PROGRAM LateBlanking_Temperature
VAR
	P3_FB_Temperature: ARRAY[1..104] OF FB_Temperature;
	i:INT;
END_VAR

ACT2();

IF Tem_HOT THEN
arrTempCtrl[1].Out.PIDRun:=TRUE;
arrTempCtrl[2].Out.PIDRun:=TRUE;
arrTempCtrl[3].Out.PIDRun:=TRUE;
arrTempCtrl[4].Out.PIDRun:=TRUE;
arrTempCtrl[5].Out.PIDRun:=TRUE;
arrTempCtrl[6].Out.PIDRun:=TRUE;
arrTempCtrl[7].Out.PIDRun:=TRUE;
arrTempCtrl[8].Out.PIDRun:=TRUE;
arrTempCtrl[9].Out.PIDRun:=TRUE;
arrTempCtrl[10].Out.PIDRun:=TRUE;
arrTempCtrl[11].Out.PIDRun:=TRUE;
arrTempCtrl[12].Out.PIDRun:=TRUE;
arrTempCtrl[13].Out.PIDRun:=TRUE;
arrTempCtrl[14].Out.PIDRun:=TRUE;
arrTempCtrl[15].Out.PIDRun:=TRUE;
arrTempCtrl[16].Out.PIDRun:=TRUE;
arrTempCtrl[17].Out.PIDRun:=TRUE;
arrTempCtrl[18].Out.PIDRun:=TRUE;
arrTempCtrl[19].Out.PIDRun:=TRUE;
arrTempCtrl[20].Out.PIDRun:=TRUE;
arrTempCtrl[21].Out.PIDRun:=TRUE;
arrTempCtrl[22].Out.PIDRun:=TRUE;
arrTempCtrl[23].Out.PIDRun:=TRUE;
arrTempCtrl[24].Out.PIDRun:=TRUE;
arrTempCtrl[25].Out.PIDRun:=TRUE;
arrTempCtrl[26].Out.PIDRun:=TRUE;
arrTempCtrl[27].Out.PIDRun:=TRUE;
arrTempCtrl[28].Out.PIDRun:=TRUE;
//arrTempCtrl[29].Out.PIDRun:=TRUE;
//arrTempCtrl[30].Out.PIDRun:=TRUE;
//arrTempCtrl[31].Out.PIDRun:=TRUE;
//arrTempCtrl[32].Out.PIDRun:=TRUE;
arrTempCtrl[33].Out.PIDRun:=TRUE;
arrTempCtrl[34].Out.PIDRun:=TRUE;
arrTempCtrl[35].Out.PIDRun:=TRUE;
arrTempCtrl[36].Out.PIDRun:=TRUE;
arrTempCtrl[37].Out.PIDRun:=TRUE;
arrTempCtrl[38].Out.PIDRun:=TRUE;
arrTempCtrl[39].Out.PIDRun:=TRUE;
arrTempCtrl[40].Out.PIDRun:=TRUE;
arrTempCtrl[41].Out.PIDRun:=TRUE;
arrTempCtrl[42].Out.PIDRun:=TRUE;
arrTempCtrl[43].Out.PIDRun:=TRUE;
arrTempCtrl[44].Out.PIDRun:=TRUE;
arrTempCtrl[45].Out.PIDRun:=TRUE;
arrTempCtrl[46].Out.PIDRun:=TRUE;
arrTempCtrl[47].Out.PIDRun:=TRUE;
arrTempCtrl[48].Out.PIDRun:=TRUE;
arrTempCtrl[49].Out.PIDRun:=TRUE;
arrTempCtrl[50].Out.PIDRun:=TRUE;
arrTempCtrl[51].Out.PIDRun:=TRUE;
arrTempCtrl[52].Out.PIDRun:=TRUE;
arrTempCtrl[53].Out.PIDRun:=TRUE;
arrTempCtrl[54].Out.PIDRun:=TRUE;
arrTempCtrl[55].Out.PIDRun:=TRUE;
arrTempCtrl[56].Out.PIDRun:=TRUE;
arrTempCtrl[57].Out.PIDRun:=TRUE;
arrTempCtrl[58].Out.PIDRun:=TRUE;
arrTempCtrl[59].Out.PIDRun:=TRUE;
arrTempCtrl[60].Out.PIDRun:=TRUE;
//arrTempCtrl[61].Out.PIDRun:=TRUE;
//arrTempCtrl[62].Out.PIDRun:=TRUE;
//arrTempCtrl[63].Out.PIDRun:=TRUE;
//arrTempCtrl[64].Out.PIDRun:=TRUE;
arrTempCtrl[65].Out.PIDRun:=TRUE;
arrTempCtrl[66].Out.PIDRun:=TRUE;
arrTempCtrl[67].Out.PIDRun:=TRUE;
arrTempCtrl[68].Out.PIDRun:=TRUE;
arrTempCtrl[69].Out.PIDRun:=TRUE;
arrTempCtrl[70].Out.PIDRun:=TRUE;
arrTempCtrl[71].Out.PIDRun:=TRUE;
arrTempCtrl[72].Out.PIDRun:=TRUE;
arrTempCtrl[73].Out.PIDRun:=TRUE;
arrTempCtrl[74].Out.PIDRun:=TRUE;
arrTempCtrl[75].Out.PIDRun:=TRUE;
arrTempCtrl[76].Out.PIDRun:=TRUE;
arrTempCtrl[77].Out.PIDRun:=TRUE;
arrTempCtrl[78].Out.PIDRun:=TRUE;
arrTempCtrl[79].Out.PIDRun:=TRUE;
arrTempCtrl[80].Out.PIDRun:=TRUE;
arrTempCtrl[81].Out.PIDRun:=TRUE;
arrTempCtrl[82].Out.PIDRun:=TRUE;
arrTempCtrl[83].Out.PIDRun:=TRUE;
arrTempCtrl[84].Out.PIDRun:=TRUE;
arrTempCtrl[85].Out.PIDRun:=TRUE;
arrTempCtrl[86].Out.PIDRun:=TRUE;
arrTempCtrl[87].Out.PIDRun:=TRUE;
arrTempCtrl[88].Out.PIDRun:=TRUE;
arrTempCtrl[89].Out.PIDRun:=TRUE;
arrTempCtrl[90].Out.PIDRun:=TRUE;
arrTempCtrl[91].Out.PIDRun:=TRUE;
arrTempCtrl[92].Out.PIDRun:=TRUE;
arrTempCtrl[93].Out.PIDRun:=TRUE;
arrTempCtrl[94].Out.PIDRun:=TRUE;
END_IF

IF Tem_Cold THEN
arrTempCtrl[1].Out.PIDRun:=FALSE;
arrTempCtrl[2].Out.PIDRun:=FALSE;
arrTempCtrl[3].Out.PIDRun:=FALSE;
arrTempCtrl[4].Out.PIDRun:=FALSE;
arrTempCtrl[5].Out.PIDRun:=FALSE;
arrTempCtrl[6].Out.PIDRun:=FALSE;
arrTempCtrl[7].Out.PIDRun:=FALSE;
arrTempCtrl[8].Out.PIDRun:=FALSE;
arrTempCtrl[9].Out.PIDRun:=FALSE;
arrTempCtrl[10].Out.PIDRun:=FALSE;
arrTempCtrl[11].Out.PIDRun:=FALSE;
arrTempCtrl[12].Out.PIDRun:=FALSE;
arrTempCtrl[13].Out.PIDRun:=FALSE;
arrTempCtrl[14].Out.PIDRun:=FALSE;
arrTempCtrl[15].Out.PIDRun:=FALSE;
arrTempCtrl[16].Out.PIDRun:=FALSE;
arrTempCtrl[17].Out.PIDRun:=FALSE;
arrTempCtrl[18].Out.PIDRun:=FALSE;
arrTempCtrl[19].Out.PIDRun:=FALSE;
arrTempCtrl[20].Out.PIDRun:=FALSE;
arrTempCtrl[21].Out.PIDRun:=FALSE;
arrTempCtrl[22].Out.PIDRun:=FALSE;
arrTempCtrl[23].Out.PIDRun:=FALSE;
arrTempCtrl[24].Out.PIDRun:=FALSE;
arrTempCtrl[25].Out.PIDRun:=FALSE;
arrTempCtrl[26].Out.PIDRun:=FALSE;
arrTempCtrl[27].Out.PIDRun:=FALSE;
arrTempCtrl[28].Out.PIDRun:=FALSE;
//arrTempCtrl[29].Out.PIDRun:=FALSE;
//arrTempCtrl[30].Out.PIDRun:=FALSE;
//arrTempCtrl[31].Out.PIDRun:=FALSE;
//arrTempCtrl[32].Out.PIDRun:=FALSE;
arrTempCtrl[33].Out.PIDRun:=FALSE;
arrTempCtrl[34].Out.PIDRun:=FALSE;
arrTempCtrl[35].Out.PIDRun:=FALSE;
arrTempCtrl[36].Out.PIDRun:=FALSE;
arrTempCtrl[37].Out.PIDRun:=FALSE;
arrTempCtrl[38].Out.PIDRun:=FALSE;
arrTempCtrl[39].Out.PIDRun:=FALSE;
arrTempCtrl[40].Out.PIDRun:=FALSE;
arrTempCtrl[41].Out.PIDRun:=FALSE;
arrTempCtrl[42].Out.PIDRun:=FALSE;
arrTempCtrl[43].Out.PIDRun:=FALSE;
arrTempCtrl[44].Out.PIDRun:=FALSE;
arrTempCtrl[45].Out.PIDRun:=FALSE;
arrTempCtrl[46].Out.PIDRun:=FALSE;
arrTempCtrl[47].Out.PIDRun:=FALSE;
arrTempCtrl[48].Out.PIDRun:=FALSE;
arrTempCtrl[49].Out.PIDRun:=FALSE;
arrTempCtrl[50].Out.PIDRun:=FALSE;
arrTempCtrl[51].Out.PIDRun:=FALSE;
arrTempCtrl[52].Out.PIDRun:=FALSE;
arrTempCtrl[53].Out.PIDRun:=FALSE;
arrTempCtrl[54].Out.PIDRun:=FALSE;
arrTempCtrl[55].Out.PIDRun:=FALSE;
arrTempCtrl[56].Out.PIDRun:=FALSE;
arrTempCtrl[57].Out.PIDRun:=FALSE;
arrTempCtrl[58].Out.PIDRun:=FALSE;
arrTempCtrl[59].Out.PIDRun:=FALSE;
arrTempCtrl[60].Out.PIDRun:=FALSE;
//arrTempCtrl[61].Out.PIDRun:=FALSE;
//arrTempCtrl[62].Out.PIDRun:=FALSE;
//arrTempCtrl[63].Out.PIDRun:=FALSE;
//arrTempCtrl[64].Out.PIDRun:=FALSE;
arrTempCtrl[65].Out.PIDRun:=FALSE;
arrTempCtrl[66].Out.PIDRun:=FALSE;
arrTempCtrl[67].Out.PIDRun:=FALSE;
arrTempCtrl[68].Out.PIDRun:=FALSE;
arrTempCtrl[69].Out.PIDRun:=FALSE;
arrTempCtrl[70].Out.PIDRun:=FALSE;
arrTempCtrl[71].Out.PIDRun:=FALSE;
arrTempCtrl[72].Out.PIDRun:=FALSE;
arrTempCtrl[73].Out.PIDRun:=FALSE;
arrTempCtrl[74].Out.PIDRun:=FALSE;
arrTempCtrl[75].Out.PIDRun:=FALSE;
arrTempCtrl[76].Out.PIDRun:=FALSE;
arrTempCtrl[77].Out.PIDRun:=FALSE;
arrTempCtrl[78].Out.PIDRun:=FALSE;
arrTempCtrl[79].Out.PIDRun:=FALSE;
arrTempCtrl[80].Out.PIDRun:=FALSE;
arrTempCtrl[81].Out.PIDRun:=FALSE;
arrTempCtrl[82].Out.PIDRun:=FALSE;
arrTempCtrl[83].Out.PIDRun:=FALSE;
arrTempCtrl[84].Out.PIDRun:=FALSE;
arrTempCtrl[85].Out.PIDRun:=FALSE;
arrTempCtrl[86].Out.PIDRun:=FALSE;
arrTempCtrl[87].Out.PIDRun:=FALSE;
arrTempCtrl[88].Out.PIDRun:=FALSE;
arrTempCtrl[89].Out.PIDRun:=FALSE;
arrTempCtrl[90].Out.PIDRun:=FALSE;
arrTempCtrl[91].Out.PIDRun:=FALSE;
arrTempCtrl[92].Out.PIDRun:=FALSE;
arrTempCtrl[93].Out.PIDRun:=FALSE;
arrTempCtrl[94].Out.PIDRun:=FALSE;
	
END_IF



//1号烤箱
IF (arrTempCtrl[1].Tem_fPV>(arrTempPar[1].fTempSet+ABS(arrTempPar[1].fTempArea)) OR arrTempCtrl[1].Tem_fPV<(arrTempPar[1].fTempSet-ABS(arrTempPar[1].fTempArea))) AND NOT P3User2_Par.Oven_Shield[1] AND P3_SystemRUN.iMode=1  THEN
	P3_Tem_Error[1]:=TRUE;//烤箱1的1板温度不在正常设定温度范围内报警
END_IF

IF (arrTempCtrl[2].Tem_fPV>(arrTempPar[2].fTempSet+ABS(arrTempPar[2].fTempArea)) OR arrTempCtrl[2].Tem_fPV<(arrTempPar[2].fTempSet-ABS(arrTempPar[2].fTempArea))) AND NOT P3User2_Par.Oven_Shield[1] AND P3_SystemRUN.iMode=1 THEN
	P3_Tem_Error[2]:=TRUE;//烤箱1的2板温度不在正常设定温度范围内报警
END_IF

IF (arrTempCtrl[3].Tem_fPV>(arrTempPar[3].fTempSet+ABS(arrTempPar[3].fTempArea)) OR arrTempCtrl[3].Tem_fPV<(arrTempPar[3].fTempSet-ABS(arrTempPar[3].fTempArea))) AND NOT P3User2_Par.Oven_Shield[1] AND P3_SystemRUN.iMode=1  THEN
	P3_Tem_Error[3]:=TRUE;//烤箱1的3板温度不在正常设定温度范围内报警
END_IF

IF (arrTempCtrl[4].Tem_fPV>(arrTempPar[4].fTempSet+ABS(arrTempPar[4].fTempArea)) OR arrTempCtrl[4].Tem_fPV<(arrTempPar[4].fTempSet-ABS(arrTempPar[4].fTempArea))) AND NOT P3User2_Par.Oven_Shield[1] AND P3_SystemRUN.iMode=1 THEN
	P3_Tem_Error[4]:=TRUE;//烤箱1的4板温度不在正常设定温度范围内报警
END_IF

//2号烤箱
IF (arrTempCtrl[5].Tem_fPV>(arrTempPar[5].fTempSet+ABS(arrTempPar[5].fTempArea)) OR arrTempCtrl[5].Tem_fPV<(arrTempPar[5].fTempSet-ABS(arrTempPar[5].fTempArea))) AND NOT P3User2_Par.Oven_Shield[4] AND P3_SystemRUN.iMode=1  THEN
	P3_Tem_Error[5]:=TRUE;//烤箱2的1板温度不在正常设定温度范围内报警
END_IF

IF (arrTempCtrl[6].Tem_fPV>(arrTempPar[6].fTempSet+ABS(arrTempPar[6].fTempArea)) OR arrTempCtrl[6].Tem_fPV<(arrTempPar[6].fTempSet-ABS(arrTempPar[6].fTempArea))) AND NOT P3User2_Par.Oven_Shield[4] AND P3_SystemRUN.iMode=1 THEN
	P3_Tem_Error[6]:=TRUE;//烤箱2的2板温度不在正常设定温度范围内报警
END_IF

IF (arrTempCtrl[7].Tem_fPV>(arrTempPar[7].fTempSet+ABS(arrTempPar[7].fTempArea)) OR arrTempCtrl[7].Tem_fPV<(arrTempPar[7].fTempSet-ABS(arrTempPar[7].fTempArea))) AND NOT P3User2_Par.Oven_Shield[4] AND P3_SystemRUN.iMode=1  THEN
	P3_Tem_Error[7]:=TRUE;//烤箱2的3板温度不在正常设定温度范围内报警
END_IF

IF (arrTempCtrl[8].Tem_fPV>(arrTempPar[8].fTempSet+ABS(arrTempPar[8].fTempArea)) OR arrTempCtrl[8].Tem_fPV<(arrTempPar[8].fTempSet-ABS(arrTempPar[8].fTempArea))) AND NOT P3User2_Par.Oven_Shield[4] AND P3_SystemRUN.iMode=1 THEN
	P3_Tem_Error[8]:=TRUE;//烤箱2的4板温度不在正常设定温度范围内报警
END_IF

//3号烤箱
IF (arrTempCtrl[9].Tem_fPV>(arrTempPar[9].fTempSet+ABS(arrTempPar[9].fTempArea)) OR arrTempCtrl[9].Tem_fPV<(arrTempPar[9].fTempSet-ABS(arrTempPar[9].fTempArea))) AND NOT P3User2_Par.Oven_Shield[7] AND P3_SystemRUN.iMode=1  THEN
	P3_Tem_Error[9]:=TRUE;//烤箱3的1板温度不在正常设定温度范围内报警
END_IF

IF (arrTempCtrl[10].Tem_fPV>(arrTempPar[10].fTempSet+ABS(arrTempPar[10].fTempArea)) OR arrTempCtrl[10].Tem_fPV<(arrTempPar[10].fTempSet-ABS(arrTempPar[10].fTempArea))) AND NOT P3User2_Par.Oven_Shield[7] AND P3_SystemRUN.iMode=1 THEN
	P3_Tem_Error[10]:=TRUE;//烤箱3的2板温度不在正常设定温度范围内报警
END_IF

IF (arrTempCtrl[11].Tem_fPV>(arrTempPar[11].fTempSet+ABS(arrTempPar[11].fTempArea)) OR arrTempCtrl[11].Tem_fPV<(arrTempPar[11].fTempSet-ABS(arrTempPar[11].fTempArea))) AND NOT P3User2_Par.Oven_Shield[7] AND P3_SystemRUN.iMode=1  THEN
	P3_Tem_Error[11]:=TRUE;//烤箱3的3板温度不在正常设定温度范围内报警
END_IF

IF (arrTempCtrl[12].Tem_fPV>(arrTempPar[12].fTempSet+ABS(arrTempPar[12].fTempArea)) OR arrTempCtrl[12].Tem_fPV<(arrTempPar[12].fTempSet-ABS(arrTempPar[12].fTempArea))) AND NOT P3User2_Par.Oven_Shield[7] AND P3_SystemRUN.iMode=1 THEN
	P3_Tem_Error[12]:=TRUE;//烤箱3的4板温度不在正常设定温度范围内报警
END_IF

//4号烤箱
IF (arrTempCtrl[13].Tem_fPV>(arrTempPar[13].fTempSet+ABS(arrTempPar[13].fTempArea)) OR arrTempCtrl[13].Tem_fPV<(arrTempPar[13].fTempSet-ABS(arrTempPar[13].fTempArea))) AND NOT P3User2_Par.Oven_Shield[10] AND P3_SystemRUN.iMode=1  THEN
	P3_Tem_Error[13]:=TRUE;//烤箱4的1板温度不在正常设定温度范围内报警
END_IF

IF (arrTempCtrl[14].Tem_fPV>(arrTempPar[14].fTempSet+ABS(arrTempPar[14].fTempArea)) OR arrTempCtrl[14].Tem_fPV<(arrTempPar[14].fTempSet-ABS(arrTempPar[14].fTempArea))) AND NOT P3User2_Par.Oven_Shield[10] AND P3_SystemRUN.iMode=1 THEN
	P3_Tem_Error[14]:=TRUE;//烤箱4的2板温度不在正常设定温度范围内报警
END_IF

IF (arrTempCtrl[15].Tem_fPV>(arrTempPar[15].fTempSet+ABS(arrTempPar[15].fTempArea)) OR arrTempCtrl[15].Tem_fPV<(arrTempPar[15].fTempSet-ABS(arrTempPar[15].fTempArea))) AND NOT P3User2_Par.Oven_Shield[10] AND P3_SystemRUN.iMode=1  THEN
	P3_Tem_Error[15]:=TRUE;//烤箱4的3板温度不在正常设定温度范围内报警
END_IF

IF (arrTempCtrl[16].Tem_fPV>(arrTempPar[16].fTempSet+ABS(arrTempPar[16].fTempArea)) OR arrTempCtrl[16].Tem_fPV<(arrTempPar[16].fTempSet-ABS(arrTempPar[16].fTempArea))) AND NOT P3User2_Par.Oven_Shield[10] AND P3_SystemRUN.iMode=1 THEN
	P3_Tem_Error[16]:=TRUE;//烤箱4的4板温度不在正常设定温度范围内报警
END_IF

//5号烤箱
IF (arrTempCtrl[17].Tem_fPV>(arrTempPar[17].fTempSet+ABS(arrTempPar[17].fTempArea)) OR arrTempCtrl[17].Tem_fPV<(arrTempPar[17].fTempSet-ABS(arrTempPar[17].fTempArea))) AND NOT P3User2_Par.Oven_Shield[13] AND P3_SystemRUN.iMode=1  THEN
	P3_Tem_Error[17]:=TRUE;//烤箱5的1板温度不在正常设定温度范围内报警
END_IF

IF (arrTempCtrl[18].Tem_fPV>(arrTempPar[18].fTempSet+ABS(arrTempPar[18].fTempArea)) OR arrTempCtrl[18].Tem_fPV<(arrTempPar[18].fTempSet-ABS(arrTempPar[18].fTempArea))) AND NOT P3User2_Par.Oven_Shield[13] AND P3_SystemRUN.iMode=1 THEN
	P3_Tem_Error[18]:=TRUE;//烤箱5的2板温度不在正常设定温度范围内报警
END_IF

IF (arrTempCtrl[19].Tem_fPV>(arrTempPar[19].fTempSet+ABS(arrTempPar[19].fTempArea)) OR arrTempCtrl[19].Tem_fPV<(arrTempPar[19].fTempSet-ABS(arrTempPar[19].fTempArea))) AND NOT P3User2_Par.Oven_Shield[13] AND P3_SystemRUN.iMode=1  THEN
	P3_Tem_Error[19]:=TRUE;//烤箱5的3板温度不在正常设定温度范围内报警
END_IF

IF (arrTempCtrl[20].Tem_fPV>(arrTempPar[20].fTempSet+ABS(arrTempPar[20].fTempArea)) OR arrTempCtrl[20].Tem_fPV<(arrTempPar[20].fTempSet-ABS(arrTempPar[20].fTempArea))) AND NOT P3User2_Par.Oven_Shield[13] AND P3_SystemRUN.iMode=1 THEN
	P3_Tem_Error[20]:=TRUE;//烤箱5的4板温度不在正常设定温度范围内报警
END_IF

//6号烤箱
IF (arrTempCtrl[21].Tem_fPV>(arrTempPar[21].fTempSet+ABS(arrTempPar[21].fTempArea)) OR arrTempCtrl[21].Tem_fPV<(arrTempPar[21].fTempSet-ABS(arrTempPar[21].fTempArea))) AND NOT P3User2_Par.Oven_Shield[16] AND P3_SystemRUN.iMode=1  THEN
	P3_Tem_Error[21]:=TRUE;//烤箱6的1板温度不在正常设定温度范围内报警
END_IF

IF (arrTempCtrl[22].Tem_fPV>(arrTempPar[22].fTempSet+ABS(arrTempPar[22].fTempArea)) OR arrTempCtrl[22].Tem_fPV<(arrTempPar[22].fTempSet-ABS(arrTempPar[22].fTempArea))) AND NOT P3User2_Par.Oven_Shield[16] AND P3_SystemRUN.iMode=1 THEN
	P3_Tem_Error[22]:=TRUE;//烤箱6的2板温度不在正常设定温度范围内报警
END_IF

IF (arrTempCtrl[23].Tem_fPV>(arrTempPar[23].fTempSet+ABS(arrTempPar[23].fTempArea)) OR arrTempCtrl[23].Tem_fPV<(arrTempPar[23].fTempSet-ABS(arrTempPar[23].fTempArea))) AND NOT P3User2_Par.Oven_Shield[16] AND P3_SystemRUN.iMode=1  THEN
	P3_Tem_Error[23]:=TRUE;//烤箱6的3板温度不在正常设定温度范围内报警
END_IF

IF (arrTempCtrl[24].Tem_fPV>(arrTempPar[24].fTempSet+ABS(arrTempPar[24].fTempArea)) OR arrTempCtrl[24].Tem_fPV<(arrTempPar[24].fTempSet-ABS(arrTempPar[24].fTempArea))) AND NOT P3User2_Par.Oven_Shield[16] AND P3_SystemRUN.iMode=1 THEN
	P3_Tem_Error[24]:=TRUE;//烤箱6的4板温度不在正常设定温度范围内报警
END_IF

//7号烤箱
IF (arrTempCtrl[25].Tem_fPV>(arrTempPar[25].fTempSet+ABS(arrTempPar[25].fTempArea)) OR arrTempCtrl[25].Tem_fPV<(arrTempPar[25].fTempSet-ABS(arrTempPar[25].fTempArea))) AND NOT P3User2_Par.Oven_Shield[19] AND P3_SystemRUN.iMode=1  THEN
	P3_Tem_Error[25]:=TRUE;//烤箱7的1板温度不在正常设定温度范围内报警
END_IF

IF (arrTempCtrl[26].Tem_fPV>(arrTempPar[26].fTempSet+ABS(arrTempPar[26].fTempArea)) OR arrTempCtrl[26].Tem_fPV<(arrTempPar[26].fTempSet-ABS(arrTempPar[26].fTempArea))) AND NOT P3User2_Par.Oven_Shield[19] AND P3_SystemRUN.iMode=1 THEN
	P3_Tem_Error[26]:=TRUE;//烤箱7的2板温度不在正常设定温度范围内报警
END_IF

IF (arrTempCtrl[27].Tem_fPV>(arrTempPar[27].fTempSet+ABS(arrTempPar[27].fTempArea)) OR arrTempCtrl[27].Tem_fPV<(arrTempPar[27].fTempSet-ABS(arrTempPar[27].fTempArea))) AND NOT P3User2_Par.Oven_Shield[19] AND P3_SystemRUN.iMode=1  THEN
	P3_Tem_Error[27]:=TRUE;//烤箱7的3板温度不在正常设定温度范围内报警
END_IF

IF (arrTempCtrl[28].Tem_fPV>(arrTempPar[28].fTempSet+ABS(arrTempPar[28].fTempArea)) OR arrTempCtrl[28].Tem_fPV<(arrTempPar[28].fTempSet-ABS(arrTempPar[28].fTempArea))) AND NOT P3User2_Par.Oven_Shield[19] AND P3_SystemRUN.iMode=1 THEN
	P3_Tem_Error[28]:=TRUE;//烤箱7的4板温度不在正常设定温度范围内报警
END_IF

//8号烤箱
IF (arrTempCtrl[33].Tem_fPV>(arrTempPar[33].fTempSet+ABS(arrTempPar[33].fTempArea)) OR arrTempCtrl[33].Tem_fPV<(arrTempPar[33].fTempSet-ABS(arrTempPar[33].fTempArea))) AND NOT P3User2_Par.Oven_Shield[2] AND P3_SystemRUN.iMode=1  THEN
	P3_Tem_Error[33]:=TRUE;//烤箱8的1板温度不在正常设定温度范围内报警
END_IF

IF (arrTempCtrl[34].Tem_fPV>(arrTempPar[34].fTempSet+ABS(arrTempPar[34].fTempArea)) OR arrTempCtrl[34].Tem_fPV<(arrTempPar[34].fTempSet-ABS(arrTempPar[34].fTempArea))) AND NOT P3User2_Par.Oven_Shield[2] AND P3_SystemRUN.iMode=1 THEN
	P3_Tem_Error[34]:=TRUE;//烤箱8的2板温度不在正常设定温度范围内报警
END_IF

IF (arrTempCtrl[35].Tem_fPV>(arrTempPar[35].fTempSet+ABS(arrTempPar[35].fTempArea)) OR arrTempCtrl[35].Tem_fPV<(arrTempPar[35].fTempSet-ABS(arrTempPar[35].fTempArea))) AND NOT P3User2_Par.Oven_Shield[2] AND P3_SystemRUN.iMode=1  THEN
	P3_Tem_Error[35]:=TRUE;//烤箱8的3板温度不在正常设定温度范围内报警
END_IF

IF (arrTempCtrl[36].Tem_fPV>(arrTempPar[36].fTempSet+ABS(arrTempPar[36].fTempArea)) OR arrTempCtrl[36].Tem_fPV<(arrTempPar[36].fTempSet-ABS(arrTempPar[36].fTempArea))) AND NOT P3User2_Par.Oven_Shield[2] AND P3_SystemRUN.iMode=1 THEN
	P3_Tem_Error[36]:=TRUE;//烤箱8的4板温度不在正常设定温度范围内报警
END_IF

//9号烤箱
IF (arrTempCtrl[37].Tem_fPV>(arrTempPar[37].fTempSet+ABS(arrTempPar[37].fTempArea)) OR arrTempCtrl[37].Tem_fPV<(arrTempPar[37].fTempSet-ABS(arrTempPar[37].fTempArea))) AND NOT P3User2_Par.Oven_Shield[5] AND P3_SystemRUN.iMode=1  THEN
	P3_Tem_Error[37]:=TRUE;//烤箱9的1板温度不在正常设定温度范围内报警
END_IF

IF (arrTempCtrl[38].Tem_fPV>(arrTempPar[38].fTempSet+ABS(arrTempPar[38].fTempArea)) OR arrTempCtrl[38].Tem_fPV<(arrTempPar[38].fTempSet-ABS(arrTempPar[38].fTempArea))) AND NOT P3User2_Par.Oven_Shield[5] AND P3_SystemRUN.iMode=1 THEN
	P3_Tem_Error[38]:=TRUE;//烤箱9的2板温度不在正常设定温度范围内报警
END_IF

IF (arrTempCtrl[39].Tem_fPV>(arrTempPar[39].fTempSet+ABS(arrTempPar[39].fTempArea)) OR arrTempCtrl[39].Tem_fPV<(arrTempPar[39].fTempSet-ABS(arrTempPar[39].fTempArea))) AND NOT P3User2_Par.Oven_Shield[5] AND P3_SystemRUN.iMode=1  THEN
	P3_Tem_Error[39]:=TRUE;//烤箱9的3板温度不在正常设定温度范围内报警
END_IF

IF (arrTempCtrl[40].Tem_fPV>(arrTempPar[40].fTempSet+ABS(arrTempPar[40].fTempArea)) OR arrTempCtrl[40].Tem_fPV<(arrTempPar[40].fTempSet-ABS(arrTempPar[40].fTempArea))) AND NOT P3User2_Par.Oven_Shield[5] AND P3_SystemRUN.iMode=1 THEN
	P3_Tem_Error[40]:=TRUE;//烤箱9的4板温度不在正常设定温度范围内报警
END_IF

//10号烤箱
IF (arrTempCtrl[41].Tem_fPV>(arrTempPar[41].fTempSet+ABS(arrTempPar[41].fTempArea)) OR arrTempCtrl[41].Tem_fPV<(arrTempPar[41].fTempSet-ABS(arrTempPar[41].fTempArea))) AND NOT P3User2_Par.Oven_Shield[8] AND P3_SystemRUN.iMode=1  THEN
	P3_Tem_Error[41]:=TRUE;//烤箱10的1板温度不在正常设定温度范围内报警
END_IF

IF (arrTempCtrl[42].Tem_fPV>(arrTempPar[42].fTempSet+ABS(arrTempPar[42].fTempArea)) OR arrTempCtrl[42].Tem_fPV<(arrTempPar[42].fTempSet-ABS(arrTempPar[42].fTempArea))) AND NOT P3User2_Par.Oven_Shield[8] AND P3_SystemRUN.iMode=1 THEN
	P3_Tem_Error[42]:=TRUE;//烤箱10的2板温度不在正常设定温度范围内报警
END_IF

IF (arrTempCtrl[43].Tem_fPV>(arrTempPar[43].fTempSet+ABS(arrTempPar[43].fTempArea)) OR arrTempCtrl[43].Tem_fPV<(arrTempPar[43].fTempSet-ABS(arrTempPar[43].fTempArea))) AND NOT P3User2_Par.Oven_Shield[8] AND P3_SystemRUN.iMode=1  THEN
	P3_Tem_Error[43]:=TRUE;//烤箱10的3板温度不在正常设定温度范围内报警
END_IF

IF (arrTempCtrl[44].Tem_fPV>(arrTempPar[44].fTempSet+ABS(arrTempPar[44].fTempArea)) OR arrTempCtrl[44].Tem_fPV<(arrTempPar[44].fTempSet-ABS(arrTempPar[44].fTempArea))) AND NOT P3User2_Par.Oven_Shield[8] AND P3_SystemRUN.iMode=1 THEN
	P3_Tem_Error[44]:=TRUE;//烤箱10的4板温度不在正常设定温度范围内报警
END_IF

//11号烤箱
IF (arrTempCtrl[45].Tem_fPV>(arrTempPar[45].fTempSet+ABS(arrTempPar[45].fTempArea)) OR arrTempCtrl[45].Tem_fPV<(arrTempPar[45].fTempSet-ABS(arrTempPar[45].fTempArea))) AND NOT P3User2_Par.Oven_Shield[11] AND P3_SystemRUN.iMode=1  THEN
	P3_Tem_Error[45]:=TRUE;//烤箱11的1板温度不在正常设定温度范围内报警
END_IF

IF (arrTempCtrl[46].Tem_fPV>(arrTempPar[46].fTempSet+ABS(arrTempPar[46].fTempArea)) OR arrTempCtrl[46].Tem_fPV<(arrTempPar[46].fTempSet-ABS(arrTempPar[46].fTempArea))) AND NOT P3User2_Par.Oven_Shield[11] AND P3_SystemRUN.iMode=1 THEN
	P3_Tem_Error[46]:=TRUE;//烤箱11的2板温度不在正常设定温度范围内报警
END_IF

IF (arrTempCtrl[47].Tem_fPV>(arrTempPar[47].fTempSet+ABS(arrTempPar[47].fTempArea)) OR arrTempCtrl[47].Tem_fPV<(arrTempPar[47].fTempSet-ABS(arrTempPar[47].fTempArea))) AND NOT P3User2_Par.Oven_Shield[11] AND P3_SystemRUN.iMode=1  THEN
	P3_Tem_Error[47]:=TRUE;//烤箱11的3板温度不在正常设定温度范围内报警
END_IF

IF (arrTempCtrl[48].Tem_fPV>(arrTempPar[48].fTempSet+ABS(arrTempPar[48].fTempArea)) OR arrTempCtrl[48].Tem_fPV<(arrTempPar[48].fTempSet-ABS(arrTempPar[48].fTempArea))) AND NOT P3User2_Par.Oven_Shield[11] AND P3_SystemRUN.iMode=1 THEN
	P3_Tem_Error[48]:=TRUE;//烤箱11的4板温度不在正常设定温度范围内报警
END_IF

//12号烤箱
IF (arrTempCtrl[49].Tem_fPV>(arrTempPar[49].fTempSet+ABS(arrTempPar[49].fTempArea)) OR arrTempCtrl[49].Tem_fPV<(arrTempPar[49].fTempSet-ABS(arrTempPar[49].fTempArea))) AND NOT P3User2_Par.Oven_Shield[14] AND P3_SystemRUN.iMode=1  THEN
	P3_Tem_Error[49]:=TRUE;//烤箱12的1板温度不在正常设定温度范围内报警
END_IF

IF (arrTempCtrl[50].Tem_fPV>(arrTempPar[50].fTempSet+ABS(arrTempPar[50].fTempArea)) OR arrTempCtrl[50].Tem_fPV<(arrTempPar[50].fTempSet-ABS(arrTempPar[50].fTempArea))) AND NOT P3User2_Par.Oven_Shield[14] AND P3_SystemRUN.iMode=1 THEN
	P3_Tem_Error[50]:=TRUE;//烤箱12的2板温度不在正常设定温度范围内报警
END_IF

IF (arrTempCtrl[51].Tem_fPV>(arrTempPar[51].fTempSet+ABS(arrTempPar[51].fTempArea)) OR arrTempCtrl[51].Tem_fPV<(arrTempPar[51].fTempSet-ABS(arrTempPar[51].fTempArea))) AND NOT P3User2_Par.Oven_Shield[14] AND P3_SystemRUN.iMode=1  THEN
	P3_Tem_Error[51]:=TRUE;//烤箱12的3板温度不在正常设定温度范围内报警
END_IF

IF (arrTempCtrl[52].Tem_fPV>(arrTempPar[52].fTempSet+ABS(arrTempPar[52].fTempArea)) OR arrTempCtrl[52].Tem_fPV<(arrTempPar[52].fTempSet-ABS(arrTempPar[52].fTempArea))) AND NOT P3User2_Par.Oven_Shield[14] AND P3_SystemRUN.iMode=1 THEN
	P3_Tem_Error[52]:=TRUE;//烤箱12的4板温度不在正常设定温度范围内报警
END_IF

//13号烤箱
IF (arrTempCtrl[53].Tem_fPV>(arrTempPar[53].fTempSet+ABS(arrTempPar[53].fTempArea)) OR arrTempCtrl[53].Tem_fPV<(arrTempPar[53].fTempSet-ABS(arrTempPar[53].fTempArea))) AND NOT P3User2_Par.Oven_Shield[17] AND P3_SystemRUN.iMode=1  THEN
	P3_Tem_Error[53]:=TRUE;//烤箱13的1板温度不在正常设定温度范围内报警
END_IF

IF (arrTempCtrl[54].Tem_fPV>(arrTempPar[54].fTempSet+ABS(arrTempPar[54].fTempArea)) OR arrTempCtrl[54].Tem_fPV<(arrTempPar[54].fTempSet-ABS(arrTempPar[54].fTempArea))) AND NOT P3User2_Par.Oven_Shield[17] AND P3_SystemRUN.iMode=1 THEN
	P3_Tem_Error[54]:=TRUE;//烤箱13的2板温度不在正常设定温度范围内报警
END_IF

IF (arrTempCtrl[55].Tem_fPV>(arrTempPar[55].fTempSet+ABS(arrTempPar[55].fTempArea)) OR arrTempCtrl[55].Tem_fPV<(arrTempPar[55].fTempSet-ABS(arrTempPar[55].fTempArea))) AND NOT P3User2_Par.Oven_Shield[17] AND P3_SystemRUN.iMode=1  THEN
	P3_Tem_Error[55]:=TRUE;//烤箱13的3板温度不在正常设定温度范围内报警
END_IF

IF (arrTempCtrl[56].Tem_fPV>(arrTempPar[56].fTempSet+ABS(arrTempPar[56].fTempArea)) OR arrTempCtrl[56].Tem_fPV<(arrTempPar[56].fTempSet-ABS(arrTempPar[56].fTempArea))) AND NOT P3User2_Par.Oven_Shield[17] AND P3_SystemRUN.iMode=1 THEN
	P3_Tem_Error[56]:=TRUE;//烤箱13的4板温度不在正常设定温度范围内报警
END_IF


//14号烤箱
IF (arrTempCtrl[57].Tem_fPV>(arrTempPar[57].fTempSet+ABS(arrTempPar[57].fTempArea)) OR arrTempCtrl[57].Tem_fPV<(arrTempPar[57].fTempSet-ABS(arrTempPar[57].fTempArea))) AND NOT P3User2_Par.Oven_Shield[20] AND P3_SystemRUN.iMode=1  THEN
	P3_Tem_Error[57]:=TRUE;//烤箱14的1板温度不在正常设定温度范围内报警
END_IF

IF (arrTempCtrl[58].Tem_fPV>(arrTempPar[58].fTempSet+ABS(arrTempPar[58].fTempArea)) OR arrTempCtrl[58].Tem_fPV<(arrTempPar[58].fTempSet-ABS(arrTempPar[58].fTempArea))) AND NOT P3User2_Par.Oven_Shield[20] AND P3_SystemRUN.iMode=1 THEN
	P3_Tem_Error[58]:=TRUE;//烤箱14的2板温度不在正常设定温度范围内报警
END_IF

IF (arrTempCtrl[59].Tem_fPV>(arrTempPar[59].fTempSet+ABS(arrTempPar[59].fTempArea)) OR arrTempCtrl[59].Tem_fPV<(arrTempPar[59].fTempSet-ABS(arrTempPar[59].fTempArea))) AND NOT P3User2_Par.Oven_Shield[20] AND P3_SystemRUN.iMode=1  THEN
	P3_Tem_Error[59]:=TRUE;//烤箱14的3板温度不在正常设定温度范围内报警
END_IF

IF (arrTempCtrl[60].Tem_fPV>(arrTempPar[60].fTempSet+ABS(arrTempPar[60].fTempArea)) OR arrTempCtrl[60].Tem_fPV<(arrTempPar[60].fTempSet-ABS(arrTempPar[60].fTempArea))) AND NOT P3User2_Par.Oven_Shield[20] AND P3_SystemRUN.iMode=1 THEN
	P3_Tem_Error[60]:=TRUE;//烤箱14的4板温度不在正常设定温度范围内报警
END_IF




//15号烤箱
IF (arrTempCtrl[65].Tem_fPV>(arrTempPar[65].fTempSet+ABS(arrTempPar[65].fTempArea)) OR arrTempCtrl[65].Tem_fPV<(arrTempPar[65].fTempSet-ABS(arrTempPar[65].fTempArea))) AND NOT P3User2_Par.Oven_Shield[3] AND P3_SystemRUN.iMode=1  THEN
	P3_Tem_Error[65]:=TRUE;//烤箱15的1板温度不在正常设定温度范围内报警
END_IF

IF (arrTempCtrl[66].Tem_fPV>(arrTempPar[66].fTempSet+ABS(arrTempPar[66].fTempArea)) OR arrTempCtrl[66].Tem_fPV<(arrTempPar[66].fTempSet-ABS(arrTempPar[66].fTempArea))) AND NOT P3User2_Par.Oven_Shield[3] AND P3_SystemRUN.iMode=1 THEN
	P3_Tem_Error[66]:=TRUE;//烤箱15的2板温度不在正常设定温度范围内报警
END_IF

IF (arrTempCtrl[67].Tem_fPV>(arrTempPar[67].fTempSet+ABS(arrTempPar[67].fTempArea)) OR arrTempCtrl[67].Tem_fPV<(arrTempPar[67].fTempSet-ABS(arrTempPar[67].fTempArea))) AND NOT P3User2_Par.Oven_Shield[3] AND P3_SystemRUN.iMode=1  THEN
	P3_Tem_Error[67]:=TRUE;//烤箱15的3板温度不在正常设定温度范围内报警
END_IF

IF (arrTempCtrl[68].Tem_fPV>(arrTempPar[68].fTempSet+ABS(arrTempPar[68].fTempArea)) OR arrTempCtrl[68].Tem_fPV<(arrTempPar[68].fTempSet-ABS(arrTempPar[68].fTempArea))) AND NOT P3User2_Par.Oven_Shield[3] AND P3_SystemRUN.iMode=1 THEN
	P3_Tem_Error[68]:=TRUE;//烤箱15的4板温度不在正常设定温度范围内报警
END_IF


//16号烤箱
IF (arrTempCtrl[69].Tem_fPV>(arrTempPar[69].fTempSet+ABS(arrTempPar[69].fTempArea)) OR arrTempCtrl[69].Tem_fPV<(arrTempPar[69].fTempSet-ABS(arrTempPar[69].fTempArea))) AND NOT P3User2_Par.Oven_Shield[6] AND P3_SystemRUN.iMode=1  THEN
	P3_Tem_Error[69]:=TRUE;//烤箱16的1板温度不在正常设定温度范围内报警
END_IF

IF (arrTempCtrl[70].Tem_fPV>(arrTempPar[70].fTempSet+ABS(arrTempPar[70].fTempArea)) OR arrTempCtrl[70].Tem_fPV<(arrTempPar[70].fTempSet-ABS(arrTempPar[70].fTempArea))) AND NOT P3User2_Par.Oven_Shield[6] AND P3_SystemRUN.iMode=1 THEN
	P3_Tem_Error[70]:=TRUE;//烤箱16的2板温度不在正常设定温度范围内报警
END_IF

IF (arrTempCtrl[71].Tem_fPV>(arrTempPar[71].fTempSet+ABS(arrTempPar[71].fTempArea)) OR arrTempCtrl[71].Tem_fPV<(arrTempPar[71].fTempSet-ABS(arrTempPar[71].fTempArea))) AND NOT P3User2_Par.Oven_Shield[6] AND P3_SystemRUN.iMode=1  THEN
	P3_Tem_Error[71]:=TRUE;//烤箱16的3板温度不在正常设定温度范围内报警
END_IF

IF (arrTempCtrl[72].Tem_fPV>(arrTempPar[72].fTempSet+ABS(arrTempPar[72].fTempArea)) OR arrTempCtrl[72].Tem_fPV<(arrTempPar[72].fTempSet-ABS(arrTempPar[72].fTempArea))) AND NOT P3User2_Par.Oven_Shield[6] AND P3_SystemRUN.iMode=1 THEN
	P3_Tem_Error[72]:=TRUE;//烤箱16的4板温度不在正常设定温度范围内报警
END_IF


//17号烤箱
IF (arrTempCtrl[73].Tem_fPV>(arrTempPar[73].fTempSet+ABS(arrTempPar[73].fTempArea)) OR arrTempCtrl[73].Tem_fPV<(arrTempPar[73].fTempSet-ABS(arrTempPar[73].fTempArea))) AND NOT P3User2_Par.Oven_Shield[9] AND P3_SystemRUN.iMode=1  THEN
	P3_Tem_Error[73]:=TRUE;//烤箱17的1板温度不在正常设定温度范围内报警
END_IF

IF (arrTempCtrl[74].Tem_fPV>(arrTempPar[74].fTempSet+ABS(arrTempPar[74].fTempArea)) OR arrTempCtrl[74].Tem_fPV<(arrTempPar[74].fTempSet-ABS(arrTempPar[74].fTempArea))) AND NOT P3User2_Par.Oven_Shield[9] AND P3_SystemRUN.iMode=1 THEN
	P3_Tem_Error[74]:=TRUE;//烤箱17的2板温度不在正常设定温度范围内报警
END_IF

IF (arrTempCtrl[75].Tem_fPV>(arrTempPar[75].fTempSet+ABS(arrTempPar[75].fTempArea)) OR arrTempCtrl[75].Tem_fPV<(arrTempPar[75].fTempSet-ABS(arrTempPar[75].fTempArea))) AND NOT P3User2_Par.Oven_Shield[9] AND P3_SystemRUN.iMode=1  THEN
	P3_Tem_Error[75]:=TRUE;//烤箱17的3板温度不在正常设定温度范围内报警
END_IF

IF (arrTempCtrl[76].Tem_fPV>(arrTempPar[76].fTempSet+ABS(arrTempPar[76].fTempArea)) OR arrTempCtrl[76].Tem_fPV<(arrTempPar[76].fTempSet-ABS(arrTempPar[76].fTempArea))) AND NOT P3User2_Par.Oven_Shield[9] AND P3_SystemRUN.iMode=1 THEN
	P3_Tem_Error[76]:=TRUE;//烤箱17的4板温度不在正常设定温度范围内报警
END_IF


//18号烤箱
IF (arrTempCtrl[77].Tem_fPV>(arrTempPar[77].fTempSet+ABS(arrTempPar[77].fTempArea)) OR arrTempCtrl[77].Tem_fPV<(arrTempPar[77].fTempSet-ABS(arrTempPar[77].fTempArea))) AND NOT P3User2_Par.Oven_Shield[12] AND P3_SystemRUN.iMode=1  THEN
	P3_Tem_Error[77]:=TRUE;//烤箱18的1板温度不在正常设定温度范围内报警
END_IF

IF (arrTempCtrl[78].Tem_fPV>(arrTempPar[78].fTempSet+ABS(arrTempPar[78].fTempArea)) OR arrTempCtrl[78].Tem_fPV<(arrTempPar[78].fTempSet-ABS(arrTempPar[78].fTempArea))) AND NOT P3User2_Par.Oven_Shield[12] AND P3_SystemRUN.iMode=1 THEN
	P3_Tem_Error[78]:=TRUE;//烤箱18的2板温度不在正常设定温度范围内报警
END_IF

IF (arrTempCtrl[79].Tem_fPV>(arrTempPar[79].fTempSet+ABS(arrTempPar[79].fTempArea)) OR arrTempCtrl[79].Tem_fPV<(arrTempPar[79].fTempSet-ABS(arrTempPar[79].fTempArea))) AND NOT P3User2_Par.Oven_Shield[12] AND P3_SystemRUN.iMode=1  THEN
	P3_Tem_Error[79]:=TRUE;//烤箱18的3板温度不在正常设定温度范围内报警
END_IF

IF (arrTempCtrl[80].Tem_fPV>(arrTempPar[80].fTempSet+ABS(arrTempPar[80].fTempArea)) OR arrTempCtrl[80].Tem_fPV<(arrTempPar[80].fTempSet-ABS(arrTempPar[80].fTempArea))) AND NOT P3User2_Par.Oven_Shield[12] AND P3_SystemRUN.iMode=1 THEN
	P3_Tem_Error[80]:=TRUE;//烤箱18的4板温度不在正常设定温度范围内报警
END_IF


//19号烤箱
IF (arrTempCtrl[81].Tem_fPV>(arrTempPar[81].fTempSet+ABS(arrTempPar[81].fTempArea)) OR arrTempCtrl[81].Tem_fPV<(arrTempPar[81].fTempSet-ABS(arrTempPar[81].fTempArea))) AND NOT P3User2_Par.Oven_Shield[15] AND P3_SystemRUN.iMode=1  THEN
	P3_Tem_Error[81]:=TRUE;//烤箱19的1板温度不在正常设定温度范围内报警
END_IF

IF (arrTempCtrl[82].Tem_fPV>(arrTempPar[82].fTempSet+ABS(arrTempPar[82].fTempArea)) OR arrTempCtrl[82].Tem_fPV<(arrTempPar[82].fTempSet-ABS(arrTempPar[82].fTempArea))) AND NOT P3User2_Par.Oven_Shield[15] AND P3_SystemRUN.iMode=1 THEN
	P3_Tem_Error[82]:=TRUE;//烤箱19的2板温度不在正常设定温度范围内报警
END_IF

IF (arrTempCtrl[83].Tem_fPV>(arrTempPar[83].fTempSet+ABS(arrTempPar[83].fTempArea)) OR arrTempCtrl[83].Tem_fPV<(arrTempPar[83].fTempSet-ABS(arrTempPar[83].fTempArea))) AND NOT P3User2_Par.Oven_Shield[15] AND P3_SystemRUN.iMode=1  THEN
	P3_Tem_Error[83]:=TRUE;//烤箱19的3板温度不在正常设定温度范围内报警
END_IF

IF (arrTempCtrl[84].Tem_fPV>(arrTempPar[84].fTempSet+ABS(arrTempPar[84].fTempArea)) OR arrTempCtrl[84].Tem_fPV<(arrTempPar[84].fTempSet-ABS(arrTempPar[84].fTempArea))) AND NOT P3User2_Par.Oven_Shield[15] AND P3_SystemRUN.iMode=1 THEN
	P3_Tem_Error[84]:=TRUE;//烤箱19的4板温度不在正常设定温度范围内报警
END_IF


//20号烤箱
IF (arrTempCtrl[85].Tem_fPV>(arrTempPar[85].fTempSet+ABS(arrTempPar[85].fTempArea)) OR arrTempCtrl[85].Tem_fPV<(arrTempPar[85].fTempSet-ABS(arrTempPar[85].fTempArea))) AND NOT P3User2_Par.Oven_Shield[18] AND P3_SystemRUN.iMode=1  THEN
	P3_Tem_Error[85]:=TRUE;//烤箱20的1板温度不在正常设定温度范围内报警
END_IF

IF (arrTempCtrl[86].Tem_fPV>(arrTempPar[86].fTempSet+ABS(arrTempPar[86].fTempArea)) OR arrTempCtrl[86].Tem_fPV<(arrTempPar[86].fTempSet-ABS(arrTempPar[86].fTempArea))) AND NOT P3User2_Par.Oven_Shield[18] AND P3_SystemRUN.iMode=1 THEN
	P3_Tem_Error[86]:=TRUE;//烤箱20的2板温度不在正常设定温度范围内报警
END_IF

IF (arrTempCtrl[87].Tem_fPV>(arrTempPar[87].fTempSet+ABS(arrTempPar[87].fTempArea)) OR arrTempCtrl[87].Tem_fPV<(arrTempPar[87].fTempSet-ABS(arrTempPar[87].fTempArea))) AND NOT P3User2_Par.Oven_Shield[18] AND P3_SystemRUN.iMode=1  THEN
	P3_Tem_Error[87]:=TRUE;//烤箱20的3板温度不在正常设定温度范围内报警
END_IF

IF (arrTempCtrl[88].Tem_fPV>(arrTempPar[88].fTempSet+ABS(arrTempPar[88].fTempArea)) OR arrTempCtrl[88].Tem_fPV<(arrTempPar[88].fTempSet-ABS(arrTempPar[88].fTempArea))) AND NOT P3User2_Par.Oven_Shield[18] AND P3_SystemRUN.iMode=1 THEN
	P3_Tem_Error[88]:=TRUE;//烤箱20的4板温度不在正常设定温度范围内报警
END_IF


//21号烤箱
IF (arrTempCtrl[89].Tem_fPV>(arrTempPar[89].fTempSet+ABS(arrTempPar[89].fTempArea)) OR arrTempCtrl[89].Tem_fPV<(arrTempPar[89].fTempSet-ABS(arrTempPar[89].fTempArea))) AND NOT P3User2_Par.Oven_Shield[21] AND P3_SystemRUN.iMode=1  THEN
	P3_Tem_Error[89]:=TRUE;//烤箱21的1板温度不在正常设定温度范围内报警
END_IF

IF (arrTempCtrl[90].Tem_fPV>(arrTempPar[90].fTempSet+ABS(arrTempPar[90].fTempArea)) OR arrTempCtrl[90].Tem_fPV<(arrTempPar[90].fTempSet-ABS(arrTempPar[90].fTempArea))) AND NOT P3User2_Par.Oven_Shield[21] AND P3_SystemRUN.iMode=1 THEN
	P3_Tem_Error[90]:=TRUE;//烤箱21的2板温度不在正常设定温度范围内报警
END_IF

IF (arrTempCtrl[91].Tem_fPV>(arrTempPar[91].fTempSet+ABS(arrTempPar[91].fTempArea)) OR arrTempCtrl[91].Tem_fPV<(arrTempPar[91].fTempSet-ABS(arrTempPar[91].fTempArea))) AND NOT P3User2_Par.Oven_Shield[21] AND P3_SystemRUN.iMode=1  THEN
	P3_Tem_Error[91]:=TRUE;//烤箱21的3板温度不在正常设定温度范围内报警
END_IF

IF (arrTempCtrl[92].Tem_fPV>(arrTempPar[92].fTempSet+ABS(arrTempPar[92].fTempArea)) OR arrTempCtrl[92].Tem_fPV<(arrTempPar[92].fTempSet-ABS(arrTempPar[92].fTempArea))) AND NOT P3User2_Par.Oven_Shield[21] AND P3_SystemRUN.iMode=1 THEN
	P3_Tem_Error[92]:=TRUE;//烤箱21的4板温度不在正常设定温度范围内报警
END_IF




//热压
IF (arrTempCtrl[93].Tem_fPV>(arrTempPar[93].fTempSet+ABS(arrTempPar[93].fTempArea)) OR arrTempCtrl[93].Tem_fPV<(arrTempPar[93].fTempSet-ABS(arrTempPar[93].fTempArea))) AND P3_SystemRUN.iMode=1  THEN
	P3_Tem_Error[93]:=TRUE;//热压上板温度不在正常设定温度范围内报警
END_IF

IF (arrTempCtrl[94].Tem_fPV>(arrTempPar[94].fTempSet+ABS(arrTempPar[94].fTempArea)) OR arrTempCtrl[94].Tem_fPV<(arrTempPar[94].fTempSet-ABS(arrTempPar[94].fTempArea))) AND P3_SystemRUN.iMode=1 THEN
	P3_Tem_Error[94]:=TRUE;//热压下板温度不在正常设定温度范围内报警
END_IF

ACTION ACT2:
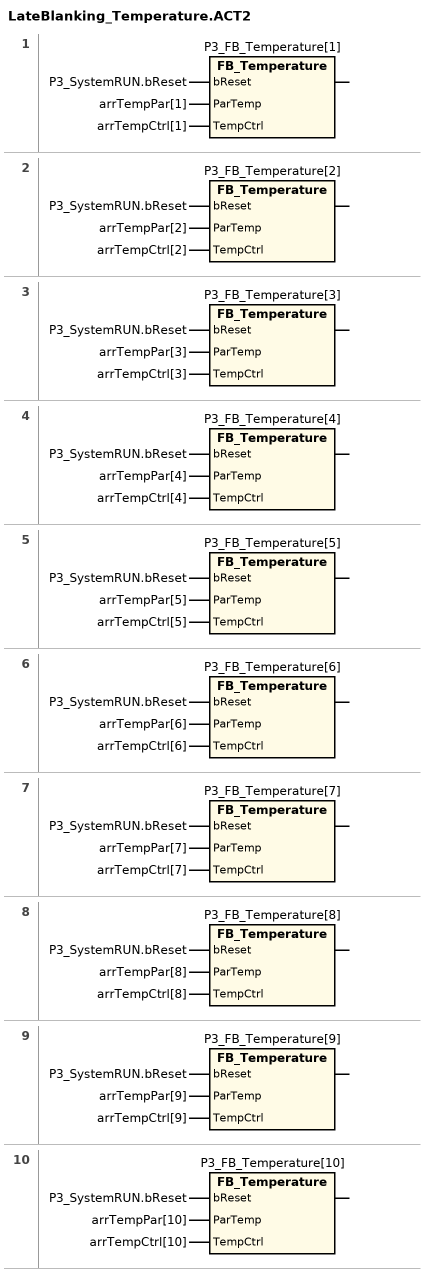
// NETWORK 1
P3_FB_Temperature[1](bReset := P3_SystemRUN.bReset, ParTemp := arrTempPar[1], TempCtrl := arrTempCtrl[1]); // FB_Temperature

// NETWORK 2
P3_FB_Temperature[2](bReset := P3_SystemRUN.bReset, ParTemp := arrTempPar[2], TempCtrl := arrTempCtrl[2]); // FB_Temperature

// NETWORK 3
P3_FB_Temperature[3](bReset := P3_SystemRUN.bReset, ParTemp := arrTempPar[3], TempCtrl := arrTempCtrl[3]); // FB_Temperature

// NETWORK 4
P3_FB_Temperature[4](bReset := P3_SystemRUN.bReset, ParTemp := arrTempPar[4], TempCtrl := arrTempCtrl[4]); // FB_Temperature

// NETWORK 5
P3_FB_Temperature[5](bReset := P3_SystemRUN.bReset, ParTemp := arrTempPar[5], TempCtrl := arrTempCtrl[5]); // FB_Temperature

// NETWORK 6
P3_FB_Temperature[6](bReset := P3_SystemRUN.bReset, ParTemp := arrTempPar[6], TempCtrl := arrTempCtrl[6]); // FB_Temperature

// NETWORK 7
P3_FB_Temperature[7](bReset := P3_SystemRUN.bReset, ParTemp := arrTempPar[7], TempCtrl := arrTempCtrl[7]); // FB_Temperature

// NETWORK 8
P3_FB_Temperature[8](bReset := P3_SystemRUN.bReset, ParTemp := arrTempPar[8], TempCtrl := arrTempCtrl[8]); // FB_Temperature

// NETWORK 9
P3_FB_Temperature[9](bReset := P3_SystemRUN.bReset, ParTemp := arrTempPar[9], TempCtrl := arrTempCtrl[9]); // FB_Temperature

// NETWORK 10
P3_FB_Temperature[10](bReset := P3_SystemRUN.bReset, ParTemp := arrTempPar[10], TempCtrl := arrTempCtrl[10]); // FB_Temperature

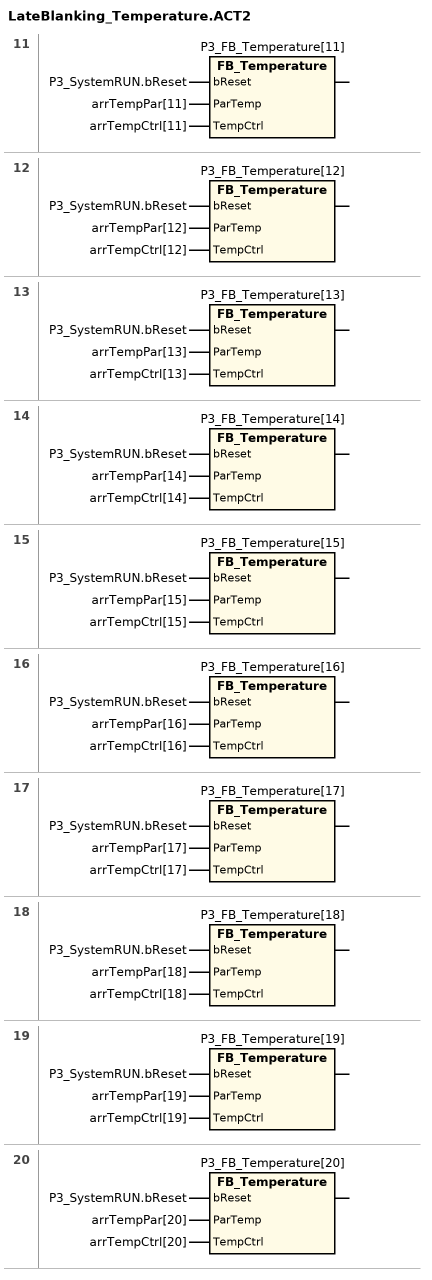
// NETWORK 11
P3_FB_Temperature[11](bReset := P3_SystemRUN.bReset, ParTemp := arrTempPar[11], TempCtrl := arrTempCtrl[11]); // FB_Temperature

// NETWORK 12
P3_FB_Temperature[12](bReset := P3_SystemRUN.bReset, ParTemp := arrTempPar[12], TempCtrl := arrTempCtrl[12]); // FB_Temperature

// NETWORK 13
P3_FB_Temperature[13](bReset := P3_SystemRUN.bReset, ParTemp := arrTempPar[13], TempCtrl := arrTempCtrl[13]); // FB_Temperature

// NETWORK 14
P3_FB_Temperature[14](bReset := P3_SystemRUN.bReset, ParTemp := arrTempPar[14], TempCtrl := arrTempCtrl[14]); // FB_Temperature

// NETWORK 15
P3_FB_Temperature[15](bReset := P3_SystemRUN.bReset, ParTemp := arrTempPar[15], TempCtrl := arrTempCtrl[15]); // FB_Temperature

// NETWORK 16
P3_FB_Temperature[16](bReset := P3_SystemRUN.bReset, ParTemp := arrTempPar[16], TempCtrl := arrTempCtrl[16]); // FB_Temperature

// NETWORK 17
P3_FB_Temperature[17](bReset := P3_SystemRUN.bReset, ParTemp := arrTempPar[17], TempCtrl := arrTempCtrl[17]); // FB_Temperature

// NETWORK 18
P3_FB_Temperature[18](bReset := P3_SystemRUN.bReset, ParTemp := arrTempPar[18], TempCtrl := arrTempCtrl[18]); // FB_Temperature

// NETWORK 19
P3_FB_Temperature[19](bReset := P3_SystemRUN.bReset, ParTemp := arrTempPar[19], TempCtrl := arrTempCtrl[19]); // FB_Temperature

// NETWORK 20
P3_FB_Temperature[20](bReset := P3_SystemRUN.bReset, ParTemp := arrTempPar[20], TempCtrl := arrTempCtrl[20]); // FB_Temperature

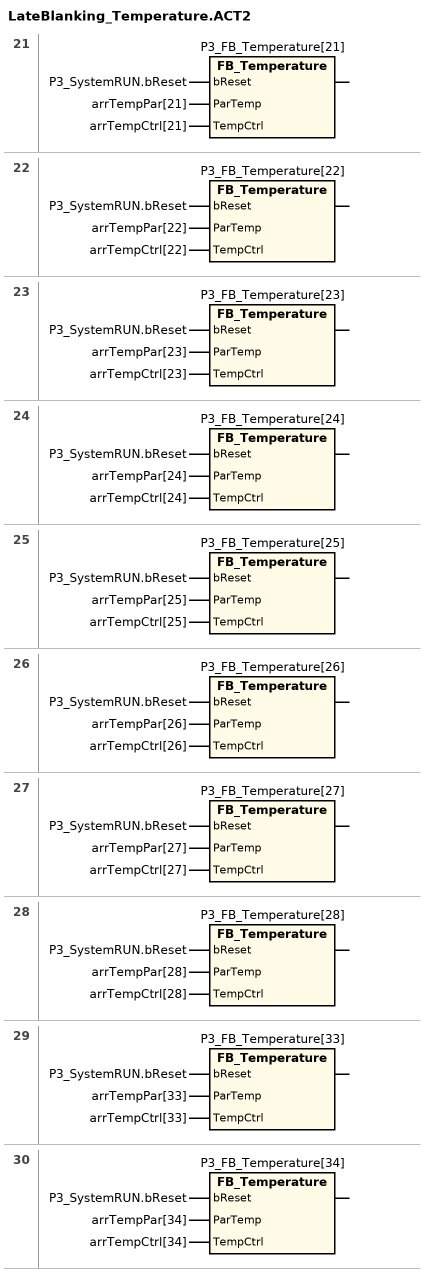
// NETWORK 21
P3_FB_Temperature[21](bReset := P3_SystemRUN.bReset, ParTemp := arrTempPar[21], TempCtrl := arrTempCtrl[21]); // FB_Temperature

// NETWORK 22
P3_FB_Temperature[22](bReset := P3_SystemRUN.bReset, ParTemp := arrTempPar[22], TempCtrl := arrTempCtrl[22]); // FB_Temperature

// NETWORK 23
P3_FB_Temperature[23](bReset := P3_SystemRUN.bReset, ParTemp := arrTempPar[23], TempCtrl := arrTempCtrl[23]); // FB_Temperature

// NETWORK 24
P3_FB_Temperature[24](bReset := P3_SystemRUN.bReset, ParTemp := arrTempPar[24], TempCtrl := arrTempCtrl[24]); // FB_Temperature

// NETWORK 25
P3_FB_Temperature[25](bReset := P3_SystemRUN.bReset, ParTemp := arrTempPar[25], TempCtrl := arrTempCtrl[25]); // FB_Temperature

// NETWORK 26
P3_FB_Temperature[26](bReset := P3_SystemRUN.bReset, ParTemp := arrTempPar[26], TempCtrl := arrTempCtrl[26]); // FB_Temperature

// NETWORK 27
P3_FB_Temperature[27](bReset := P3_SystemRUN.bReset, ParTemp := arrTempPar[27], TempCtrl := arrTempCtrl[27]); // FB_Temperature

// NETWORK 28
P3_FB_Temperature[28](bReset := P3_SystemRUN.bReset, ParTemp := arrTempPar[28], TempCtrl := arrTempCtrl[28]); // FB_Temperature

// NETWORK 29
P3_FB_Temperature[33](bReset := P3_SystemRUN.bReset, ParTemp := arrTempPar[33], TempCtrl := arrTempCtrl[33]); // FB_Temperature

// NETWORK 30
P3_FB_Temperature[34](bReset := P3_SystemRUN.bReset, ParTemp := arrTempPar[34], TempCtrl := arrTempCtrl[34]); // FB_Temperature

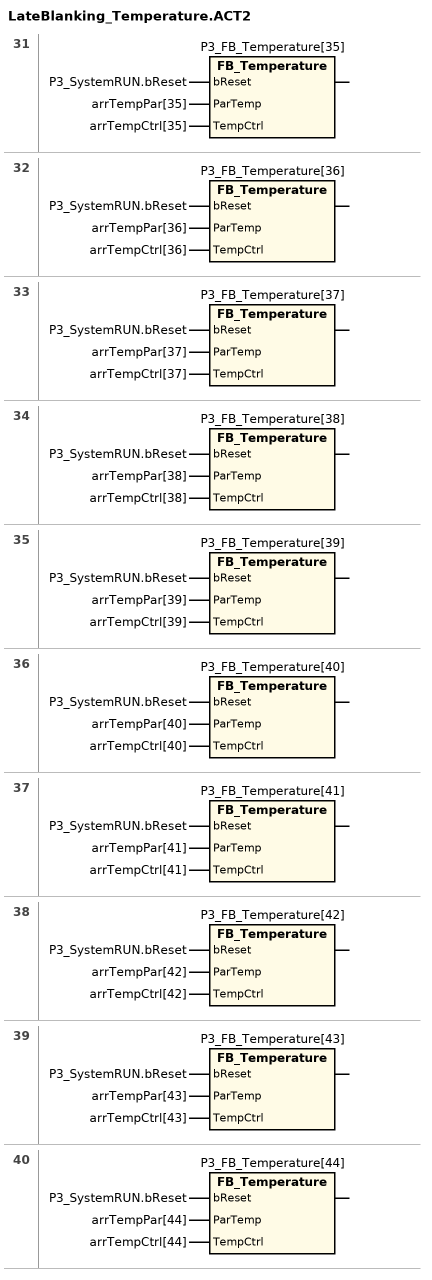
// NETWORK 31
P3_FB_Temperature[35](bReset := P3_SystemRUN.bReset, ParTemp := arrTempPar[35], TempCtrl := arrTempCtrl[35]); // FB_Temperature

// NETWORK 32
P3_FB_Temperature[36](bReset := P3_SystemRUN.bReset, ParTemp := arrTempPar[36], TempCtrl := arrTempCtrl[36]); // FB_Temperature

// NETWORK 33
P3_FB_Temperature[37](bReset := P3_SystemRUN.bReset, ParTemp := arrTempPar[37], TempCtrl := arrTempCtrl[37]); // FB_Temperature

// NETWORK 34
P3_FB_Temperature[38](bReset := P3_SystemRUN.bReset, ParTemp := arrTempPar[38], TempCtrl := arrTempCtrl[38]); // FB_Temperature

// NETWORK 35
P3_FB_Temperature[39](bReset := P3_SystemRUN.bReset, ParTemp := arrTempPar[39], TempCtrl := arrTempCtrl[39]); // FB_Temperature

// NETWORK 36
P3_FB_Temperature[40](bReset := P3_SystemRUN.bReset, ParTemp := arrTempPar[40], TempCtrl := arrTempCtrl[40]); // FB_Temperature

// NETWORK 37
P3_FB_Temperature[41](bReset := P3_SystemRUN.bReset, ParTemp := arrTempPar[41], TempCtrl := arrTempCtrl[41]); // FB_Temperature

// NETWORK 38
P3_FB_Temperature[42](bReset := P3_SystemRUN.bReset, ParTemp := arrTempPar[42], TempCtrl := arrTempCtrl[42]); // FB_Temperature

// NETWORK 39
P3_FB_Temperature[43](bReset := P3_SystemRUN.bReset, ParTemp := arrTempPar[43], TempCtrl := arrTempCtrl[43]); // FB_Temperature

// NETWORK 40
P3_FB_Temperature[44](bReset := P3_SystemRUN.bReset, ParTemp := arrTempPar[44], TempCtrl := arrTempCtrl[44]); // FB_Temperature

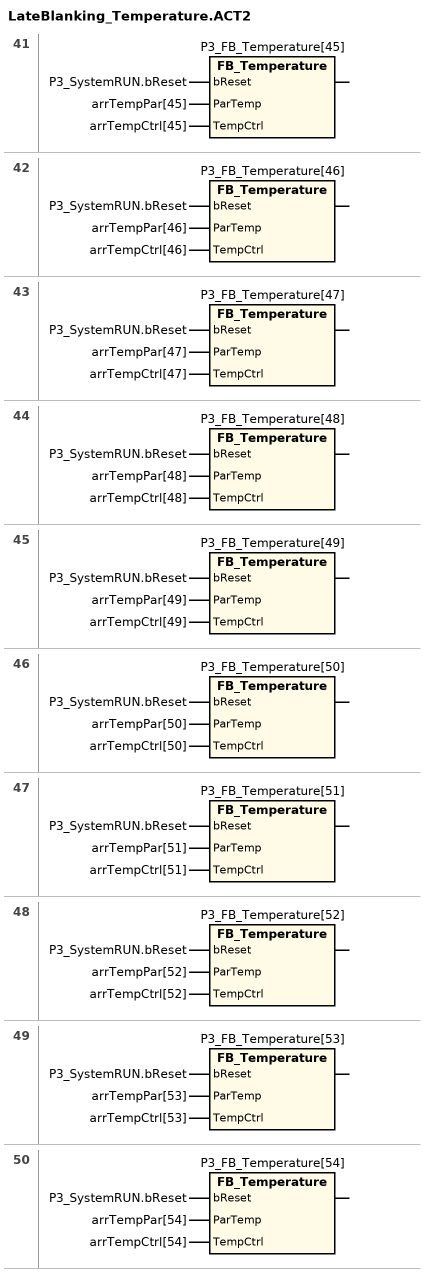
// NETWORK 41
P3_FB_Temperature[45](bReset := P3_SystemRUN.bReset, ParTemp := arrTempPar[45], TempCtrl := arrTempCtrl[45]); // FB_Temperature

// NETWORK 42
P3_FB_Temperature[46](bReset := P3_SystemRUN.bReset, ParTemp := arrTempPar[46], TempCtrl := arrTempCtrl[46]); // FB_Temperature

// NETWORK 43
P3_FB_Temperature[47](bReset := P3_SystemRUN.bReset, ParTemp := arrTempPar[47], TempCtrl := arrTempCtrl[47]); // FB_Temperature

// NETWORK 44
P3_FB_Temperature[48](bReset := P3_SystemRUN.bReset, ParTemp := arrTempPar[48], TempCtrl := arrTempCtrl[48]); // FB_Temperature

// NETWORK 45
P3_FB_Temperature[49](bReset := P3_SystemRUN.bReset, ParTemp := arrTempPar[49], TempCtrl := arrTempCtrl[49]); // FB_Temperature

// NETWORK 46
P3_FB_Temperature[50](bReset := P3_SystemRUN.bReset, ParTemp := arrTempPar[50], TempCtrl := arrTempCtrl[50]); // FB_Temperature

// NETWORK 47
P3_FB_Temperature[51](bReset := P3_SystemRUN.bReset, ParTemp := arrTempPar[51], TempCtrl := arrTempCtrl[51]); // FB_Temperature

// NETWORK 48
P3_FB_Temperature[52](bReset := P3_SystemRUN.bReset, ParTemp := arrTempPar[52], TempCtrl := arrTempCtrl[52]); // FB_Temperature

// NETWORK 49
P3_FB_Temperature[53](bReset := P3_SystemRUN.bReset, ParTemp := arrTempPar[53], TempCtrl := arrTempCtrl[53]); // FB_Temperature

// NETWORK 50
P3_FB_Temperature[54](bReset := P3_SystemRUN.bReset, ParTemp := arrTempPar[54], TempCtrl := arrTempCtrl[54]); // FB_Temperature

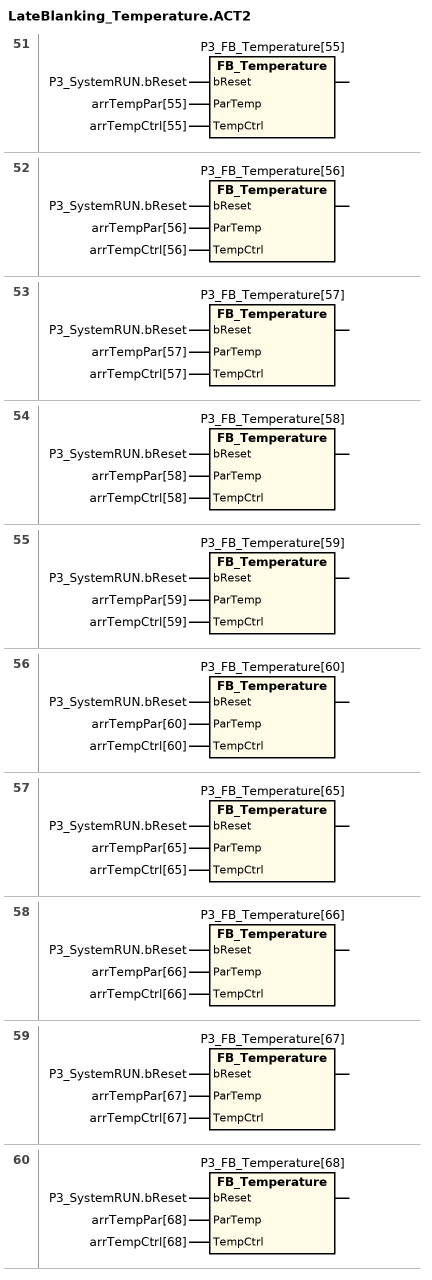
// NETWORK 51
P3_FB_Temperature[55](bReset := P3_SystemRUN.bReset, ParTemp := arrTempPar[55], TempCtrl := arrTempCtrl[55]); // FB_Temperature

// NETWORK 52
P3_FB_Temperature[56](bReset := P3_SystemRUN.bReset, ParTemp := arrTempPar[56], TempCtrl := arrTempCtrl[56]); // FB_Temperature

// NETWORK 53
P3_FB_Temperature[57](bReset := P3_SystemRUN.bReset, ParTemp := arrTempPar[57], TempCtrl := arrTempCtrl[57]); // FB_Temperature

// NETWORK 54
P3_FB_Temperature[58](bReset := P3_SystemRUN.bReset, ParTemp := arrTempPar[58], TempCtrl := arrTempCtrl[58]); // FB_Temperature

// NETWORK 55
P3_FB_Temperature[59](bReset := P3_SystemRUN.bReset, ParTemp := arrTempPar[59], TempCtrl := arrTempCtrl[59]); // FB_Temperature

// NETWORK 56
P3_FB_Temperature[60](bReset := P3_SystemRUN.bReset, ParTemp := arrTempPar[60], TempCtrl := arrTempCtrl[60]); // FB_Temperature

// NETWORK 57
P3_FB_Temperature[65](bReset := P3_SystemRUN.bReset, ParTemp := arrTempPar[65], TempCtrl := arrTempCtrl[65]); // FB_Temperature

// NETWORK 58
P3_FB_Temperature[66](bReset := P3_SystemRUN.bReset, ParTemp := arrTempPar[66], TempCtrl := arrTempCtrl[66]); // FB_Temperature

// NETWORK 59
P3_FB_Temperature[67](bReset := P3_SystemRUN.bReset, ParTemp := arrTempPar[67], TempCtrl := arrTempCtrl[67]); // FB_Temperature

// NETWORK 60
P3_FB_Temperature[68](bReset := P3_SystemRUN.bReset, ParTemp := arrTempPar[68], TempCtrl := arrTempCtrl[68]); // FB_Temperature

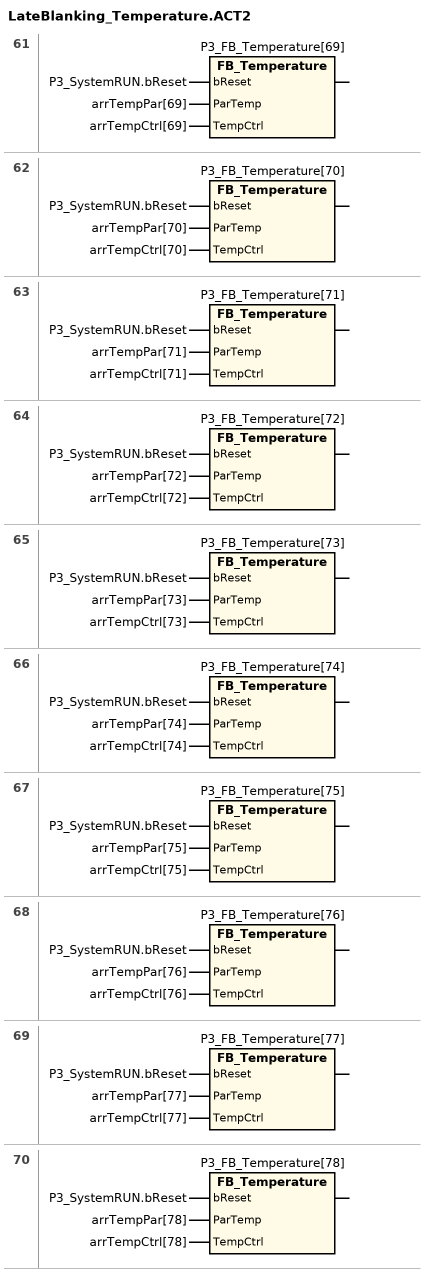
// NETWORK 61
P3_FB_Temperature[69](bReset := P3_SystemRUN.bReset, ParTemp := arrTempPar[69], TempCtrl := arrTempCtrl[69]); // FB_Temperature

// NETWORK 62
P3_FB_Temperature[70](bReset := P3_SystemRUN.bReset, ParTemp := arrTempPar[70], TempCtrl := arrTempCtrl[70]); // FB_Temperature

// NETWORK 63
P3_FB_Temperature[71](bReset := P3_SystemRUN.bReset, ParTemp := arrTempPar[71], TempCtrl := arrTempCtrl[71]); // FB_Temperature

// NETWORK 64
P3_FB_Temperature[72](bReset := P3_SystemRUN.bReset, ParTemp := arrTempPar[72], TempCtrl := arrTempCtrl[72]); // FB_Temperature

// NETWORK 65
P3_FB_Temperature[73](bReset := P3_SystemRUN.bReset, ParTemp := arrTempPar[73], TempCtrl := arrTempCtrl[73]); // FB_Temperature

// NETWORK 66
P3_FB_Temperature[74](bReset := P3_SystemRUN.bReset, ParTemp := arrTempPar[74], TempCtrl := arrTempCtrl[74]); // FB_Temperature

// NETWORK 67
P3_FB_Temperature[75](bReset := P3_SystemRUN.bReset, ParTemp := arrTempPar[75], TempCtrl := arrTempCtrl[75]); // FB_Temperature

// NETWORK 68
P3_FB_Temperature[76](bReset := P3_SystemRUN.bReset, ParTemp := arrTempPar[76], TempCtrl := arrTempCtrl[76]); // FB_Temperature

// NETWORK 69
P3_FB_Temperature[77](bReset := P3_SystemRUN.bReset, ParTemp := arrTempPar[77], TempCtrl := arrTempCtrl[77]); // FB_Temperature

// NETWORK 70
P3_FB_Temperature[78](bReset := P3_SystemRUN.bReset, ParTemp := arrTempPar[78], TempCtrl := arrTempCtrl[78]); // FB_Temperature

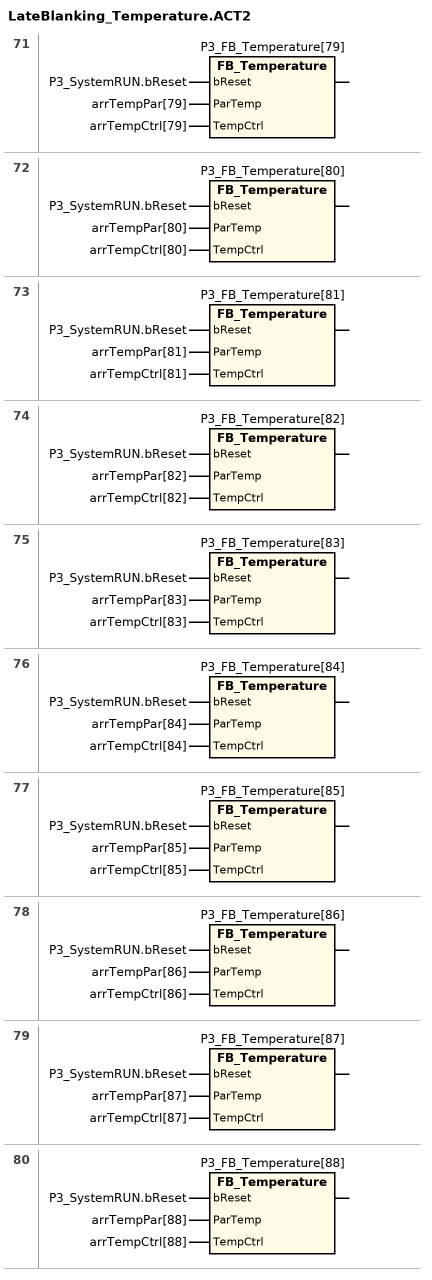
// NETWORK 71
P3_FB_Temperature[79](bReset := P3_SystemRUN.bReset, ParTemp := arrTempPar[79], TempCtrl := arrTempCtrl[79]); // FB_Temperature

// NETWORK 72
P3_FB_Temperature[80](bReset := P3_SystemRUN.bReset, ParTemp := arrTempPar[80], TempCtrl := arrTempCtrl[80]); // FB_Temperature

// NETWORK 73
P3_FB_Temperature[81](bReset := P3_SystemRUN.bReset, ParTemp := arrTempPar[81], TempCtrl := arrTempCtrl[81]); // FB_Temperature

// NETWORK 74
P3_FB_Temperature[82](bReset := P3_SystemRUN.bReset, ParTemp := arrTempPar[82], TempCtrl := arrTempCtrl[82]); // FB_Temperature

// NETWORK 75
P3_FB_Temperature[83](bReset := P3_SystemRUN.bReset, ParTemp := arrTempPar[83], TempCtrl := arrTempCtrl[83]); // FB_Temperature

// NETWORK 76
P3_FB_Temperature[84](bReset := P3_SystemRUN.bReset, ParTemp := arrTempPar[84], TempCtrl := arrTempCtrl[84]); // FB_Temperature

// NETWORK 77
P3_FB_Temperature[85](bReset := P3_SystemRUN.bReset, ParTemp := arrTempPar[85], TempCtrl := arrTempCtrl[85]); // FB_Temperature

// NETWORK 78
P3_FB_Temperature[86](bReset := P3_SystemRUN.bReset, ParTemp := arrTempPar[86], TempCtrl := arrTempCtrl[86]); // FB_Temperature

// NETWORK 79
P3_FB_Temperature[87](bReset := P3_SystemRUN.bReset, ParTemp := arrTempPar[87], TempCtrl := arrTempCtrl[87]); // FB_Temperature

// NETWORK 80
P3_FB_Temperature[88](bReset := P3_SystemRUN.bReset, ParTemp := arrTempPar[88], TempCtrl := arrTempCtrl[88]); // FB_Temperature

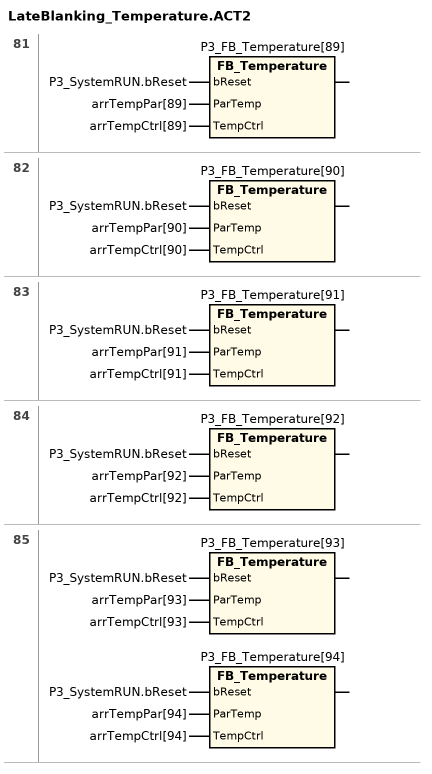
// NETWORK 81
P3_FB_Temperature[89](bReset := P3_SystemRUN.bReset, ParTemp := arrTempPar[89], TempCtrl := arrTempCtrl[89]); // FB_Temperature

// NETWORK 82
P3_FB_Temperature[90](bReset := P3_SystemRUN.bReset, ParTemp := arrTempPar[90], TempCtrl := arrTempCtrl[90]); // FB_Temperature

// NETWORK 83
P3_FB_Temperature[91](bReset := P3_SystemRUN.bReset, ParTemp := arrTempPar[91], TempCtrl := arrTempCtrl[91]); // FB_Temperature

// NETWORK 84
P3_FB_Temperature[92](bReset := P3_SystemRUN.bReset, ParTemp := arrTempPar[92], TempCtrl := arrTempCtrl[92]); // FB_Temperature

// NETWORK 85
P3_FB_Temperature[93](bReset := P3_SystemRUN.bReset, ParTemp := arrTempPar[93], TempCtrl := arrTempCtrl[93]); // FB_Temperature
P3_FB_Temperature[94](bReset := P3_SystemRUN.bReset, ParTemp := arrTempPar[94], TempCtrl := arrTempCtrl[94]); // FB_Temperature
END_ACTION

END_PROGRAM

(* stored: Version 1.1.0.1, ProductVersion 3.1.4024.12
   POU LateBlanking_Temperature: Id {9bd96bdd-7f05-4453-ad0a-e07670b1ef1d}, SpecialFunc None
   Action ACT2: Id {b7862ffb-3437-4717-b9bd-66eff8a18c40} *)
